TYPE typeMotionSide :
STRUCT
	RequestCoil: BOOL;		//TRUE if the coil to advance the motion has been switched on
	Depth: BOOL;  			//TRUE if the motion is complete
	Prompt: BOOL;           //TRUE if the motion is OK to move (or to the next step)
	InterlockOK: BOOL;		//TRUE if the interlock is satisified for the motion
	NumberOrder:UINT;		//number of the motion to take

	TimeTaken: TIME;		//Time Taken for the motion to complete
	
	valCoil: INT := 1;		
	valDepth: INT := 2;
	
	bHideCoil: BOOL;		//TRUE to hide the coil
	bHideDepth: BOOL;		//TRUE to hide the depth
	bHideInterlock: BOOL;	//TRUE to hide the interlock
	bHidePrompt: BOOL;		//TRUE to hide the prompt
	bHideTime: BOOL;		//TRUE to hide the time
	bHideButton: BOOL;		//TRUE to hide the button
	
	FdbkColour: DWORD := 16#FFC6C6C6; //sensor feedback colour
	CoilColour:DWORD := 16#FFC6C6C6; //coil feedback colour


END_STRUCT
END_TYPE

(* stored: Version 1.1.0.1, ProductVersion 3.1.4024.12
   DUT typeMotionSide: Id {80cb6d72-5b27-4fe2-bda0-dfb325271228} *)
